Universal Robots PolyScope program: v2.5ross.urp

Program v2.5ross (installation=botross directory=/programs/usbdisk/APS2OsUltimosRomanticos createdIn=3.15.3.106223 lastSavedIn=3.15.3.106223 robotSerialNumber=2017357016)
Calibrated DH parameters: a=[0.000147, -0.403633, -0.391058, 0.000042, 0.000118, 0]; d=[0.089178, 30.14366, -33.809995, 3.776935, 0.094786, 0.082481]; alpha=[1.56929, -0.004446, 0.00863, 1.569893, -1.570304, 0]; deltaTheta=[0.000049, -0.320568, 0.239888, 0.08077, 0.000061, 0.000065]
BeforeStart
  Socket_ready := True
  Z := 0
  Socket := socket_open("10.103.16.11",20000)
  Socket_color := socket_open("10.103.16.11",30000)
  Num_points := socket_read_ascii_float(1)
  PosicaoRecarga := 1
  posicao_tinta := p[15*PosicaoRecarga/1000,(PosicaoRecarga+7)/7*15/1000,0,0,0,0]
  Recarga := False
  MoveL speed 250 mm/s, acceleration 1200 mm/s^2 (useActiveTCP=true) feature=Plano_Tintas
    Waypoint Waypoint (Variable): variable=posicao_tinta
Robot Program (runOnlyOnce=false)
  If Socket_ready ≟  True
    Loop While (checkContinuously=false) expression=Socket≟ False
      Socket := socket_open("10.103.16.11",20000)
    Num_points := socket_read_ascii_float(1)
    N := Num_points[1]
    X := socket_read_ascii_float(N)
    Y := socket_read_ascii_float(N)
    Z := socket_read_ascii_float(N)
    Socket_ready := False
  SuppressedNode
    Socket := socket_close()
  count := 1
  If Recarga ≟ False
    Loop While (checkContinuously=false) expression=count≤N
      move2pose := p[X[count]/1000,Y[count]/1000,Z[count]/1000,0,0,0]
      MoveL speed 200 mm/s, acceleration 600 mm/s^2 (useActiveTCP=true) feature=Plano_Pintura
        Waypoint Waypoint (Variable): variable=move2pose
      SuppressedNode
        Wait Sleep waitTime=0.5
      count := count+1
  If Recarga ≟  True
    MoveL speed 250 mm/s, acceleration 1200 mm/s^2 (useActiveTCP=true) feature=Plano_Tintas
      Waypoint Waypoint (Variable): variable=posicao_tinta
    Recarga := False
  SuppressedNode
    Script: socket_close()
Thread Thread_1 (runOnlyOnce=false)
  Wait Sleep waitTime=60
  Recarga := True
  posicao_tinta := p[15*PosicaoRecarga/1000,PosicaoRecarga/7*15/1000,0,0,0,0]
Thread Thread_2 (runOnlyOnce=false)
  SuppressedNode
    Loop While (checkContinuously=false) expression=Socket≟ False
      Socket := socket_open("10.103.16.11",30000)
  If Z ≟ 120
    Wait Sleep waitTime=10
    Socket_ready := True
